DATA_BLOCK "bioAct.DB"
{ S7_Optimized_Access := 'TRUE' }
VERSION : 1.0
// Batch I/O Actuator Data Block:
// by Woermann Automation
NON_RETAIN
   VAR RETAIN
      Act : Array[0..15] of "bioAct.DT";
   END_VAR

BEGIN

END_DATA_BLOCK

